{attribute 'linkalways'}
{attribute 'no_explicit_call' := 'This FB is a CLASS and must be accessed using methods or properties'}
{attribute 'enable_dynamic_creation'}
FUNCTION_BLOCK _ETcVnDotCodeOptions EXTENDS EnumDatatypeBase
VAR
	localData : ETcVnDotCodeOptions;
	activeData : REFERENCE TO ETcVnDotCodeOptions;
	enumBaseDatatype : _ULINT(localData);
END_VAR

METHOD PRIVATE AddLocalEnumeration
VAR_INPUT
	Enumeration : T_MAXSTRING;
	Value : ETcVnDotCodeOptions;
END_VAR
AddEnumeration(Enumeration, Value);
END_METHOD

PROPERTY PUBLIC Address : PVOID
GET
Address := ADR(activeData);
END_GET
END_PROPERTY

METHOD PUBLIC ClearReference
VAR_INPUT
END_VAR
activeData REF= localData;
SetBaseDatatypeReference();
END_METHOD

METHOD PUBLIC Clone : I_Datatype
VAR
    pClone : POINTER TO _ETcVnDotCodeOptions;
END_VAR
pClone := __NEW(_ETcVnDotCodeOptions(InitialValue := Value));
IF pClone = 0 THEN
    RETURN;
END_IF
Clone := pClone^;
END_METHOD

METHOD FB_init : BOOL
VAR_INPUT
	bInitRetains : BOOL; // if TRUE, the retain variables are initialized (warm start / cold start)
	bInCopyCode : BOOL;  // if TRUE, the instance afterwards gets moved into the copy code (online change)
	InitialValue : ETcVnDotCodeOptions;
END_VAR
localData := InitialValue;
AddBaseDatatype(enumBaseDatatype);
ClearReference();

AddLocalEnumeration('TCVN_DCO_DEFAULT', ETcVnDotCodeOptions.TCVN_DCO_DEFAULT);
AddLocalEnumeration('TCVN_DCO_BINARY_INPUT', ETcVnDotCodeOptions.TCVN_DCO_BINARY_INPUT);
AddLocalEnumeration('TCVN_DCO_DETECTBLOBS', ETcVnDotCodeOptions.TCVN_DCO_DETECTBLOBS);
AddLocalEnumeration('TCVN_DCO_FILTERCONTOURS', ETcVnDotCodeOptions.TCVN_DCO_FILTERCONTOURS);
AddLocalEnumeration('TCVN_DCO_REGULAR_COLOR', ETcVnDotCodeOptions.TCVN_DCO_REGULAR_COLOR);
AddLocalEnumeration('TCVN_DCO_INVERTED_COLOR', ETcVnDotCodeOptions.TCVN_DCO_INVERTED_COLOR);
END_METHOD

PROPERTY PUBLIC Identifier : T_MAXSTRING
GET
Identifier := 'ETcVnDotCodeOptions';
END_GET
END_PROPERTY

METHOD IsEnumeratorValueEqual : BOOL
VAR_INPUT
	Enumerator : I_KeyValueForwardEnumerator;
END_VAR
VAR
	storedValue : ETcVnDotCodeOptions;
END_VAR
IF NOT Enumerator.TryGet(storedValue) THEN
	RETURN;
END_IF

IsEnumeratorValueEqual := storedValue = activeData;
END_METHOD

METHOD PUBLIC MakeReferenceTo
VAR_INPUT
	ReferenceTarget : REFERENCE TO ETcVnDotCodeOptions;
END_VAR
activeData REF= ReferenceTarget;
SetBaseDatatypeReference();
END_METHOD

METHOD PROTECTED SetBaseDatatypeReference
VAR_INPUT
END_VAR
enumBaseDatatype.MakeReferenceTo(activeData);
END_METHOD

PROPERTY PUBLIC Size : UDINT
GET
Size := SIZEOF(activeData);
END_GET
END_PROPERTY

METHOD TryMakeReferenceTo : BOOL
VAR_INPUT
	Target : I_Datatype;
END_VAR
VAR
	pTargetData : POINTER TO ETcVnDotCodeOptions;
END_VAR
IF NOT IsEquivalentTo(Target) THEN
	RETURN;
END_IF

pTargetData := Target.Address;
activeData REF= pTargetData^;
SetBaseDatatypeReference();
TryMakeReferenceTo := TRUE;
END_METHOD

PROPERTY PUBLIC Value : ETcVnDotCodeOptions
GET
Value := activeData;
END_GET
SET
activeData := Value;
END_SET
END_PROPERTY

END_FUNCTION_BLOCK

(* stored: Version 1.1.0.1, ProductVersion 3.1.4026.13
   POU _ETcVnDotCodeOptions: Id {8395b0b9-90b2-4cb3-a40f-690645cbb571}, SpecialFunc None
   Folder Core: Id {0f8e67ae-07f5-4d86-b018-5069aaa45fe2}
   Folder Protected: Id {5d76298d-b914-41dc-9e1d-736b7932f759}
   Folder Customize: Id {2c5b5cb7-95be-4998-9d2f-d63d43103e0c}
   Folder Constructor: Id {f4da4b9f-147f-4d4b-bb19-52e7dea686f7}
   Folder Private: Id {99246adc-7415-45fc-a78e-8831f633e1bb}
   Folder Protected: Id {d0241f52-3e4a-47a8-a793-d2960f92771c}
   Method AddLocalEnumeration: Id {b467e7df-3d1f-4dcf-a708-21cbfd55df9e}
   Property Address: Id {4de887d7-4aff-49ed-9ece-663918dc5db7}
   Get Get: Id {d486bc6b-fb7d-4a51-adcf-9d16c0f1a60e}
   Method ClearReference: Id {5a2d8fdf-5314-487e-99b6-7368725c3850}
   Method Clone: Id {cc700985-a958-4c14-8e98-39b36d02438c}
   Method FB_init: Id {ced9d9d2-7455-4f43-915a-773dc60bbe96}
   Property Identifier: Id {c2cf669f-4024-4de8-82b9-1cca0f5eeb2d}
   Get Get: Id {c9a08d9a-7587-4fbc-9069-4ca536cc01da}
   Method IsEnumeratorValueEqual: Id {7718c76d-1992-49b3-8935-70de3a6ab3c3}
   Method MakeReferenceTo: Id {d1e2e7eb-1494-449d-a3a3-bf0c88e3a345}
   Method SetBaseDatatypeReference: Id {767231be-5c5e-40cd-a208-e95677df3bfe}
   Property Size: Id {527cef61-834f-496d-ab86-0c6ae8fcc2a7}
   Get Get: Id {6244f4e1-4ce7-411f-805e-443100b50b6a}
   Method TryMakeReferenceTo: Id {fb289bef-cbab-4a76-aba3-d69ba0e434a9}
   Property Value: Id {c1b238ba-0fd8-4b8b-9d5b-adb74ad7b540}
   Get Get: Id {e22c546d-af09-4e59-9818-1ee2d42c321f}
   Set Set: Id {d5bdff57-56be-43c8-999a-c19657f27924} *)
